FUNCTION_BLOCK Testowy3
VAR
	bTest3: BOOL;
END_VAR

END_FUNCTION_BLOCK

(* stored: Version 1.1.0.1
   POU Testowy3: Id {4577185b-52ff-4094-ab7e-f3269012a1ad}, SpecialFunc None *)
